(* IEC 61131-3 sources: Lasal/CPU_5344_V01/Class/MillPlanes, 1 file *)

(* ---- MillPlanes.st ---- *)
(*!
<Class
	Name               = "MillPlanes"
	Revision           = "0.0"
	RealtimeTask       = "false"
	CyclicTask         = "false"
	BackgroundTask     = "false"
	Sigmatek           = "false"
	OSInterface        = "false"
	HighPriority       = "false"
	Automatic          = "false"
	UpdateMode         = "Prescan"
	SharedCommandTable = "true"
	Objectsize         = "(450,120)">
	<Channels>
		<Server Name="ClassSvr" Visualized="false" Initialize="false" WriteProtected="true" Retentive="false"/>
		<Server Name="firstIdx" Visualized="true" Initialize="false" WriteProtected="false" Retentive="false"/>
		<Client Name="Line1" Required="true" Internal="true"/>
		<Client Name="Line2" Required="true" Internal="true"/>
		<Client Name="Line3" Required="true" Internal="true"/>
		<Client Name="Line4" Required="true" Internal="true"/>
		<Client Name="Line5" Required="true" Internal="true"/>
		<Client Name="Line6" Required="true" Internal="true"/>
	</Channels>
	<Network Name="MillPlanes">
		<!-- List of Components in this network -->
		<Components>
			<Object
				Name       = "Line1"
				Class      = "MillPlane"
				Position   = "(150,270)"
				Visualized = "true">
				<Channels>
					<Server Name="amount"/>
					<Server Name="ClassSvr"/>
					<Server Name="depth"/>
					<Server Name="feedRate"/>
					<Server Name="firsIdx"/>
					<Server Name="lowerRate"/>
					<Server Name="rnr"/>
				</Channels>
			</Object>
			<Object
				Name       = "Line2"
				Class      = "MillPlane"
				Position   = "(690,270)"
				Visualized = "true">
				<Channels>
					<Server Name="amount"/>
					<Server Name="ClassSvr"/>
					<Server Name="depth"/>
					<Server Name="feedRate"/>
					<Server Name="firsIdx"/>
					<Server Name="lowerRate"/>
					<Server Name="rnr"/>
				</Channels>
			</Object>
			<Object
				Name       = "Line3"
				Class      = "MillPlane"
				Position   = "(1230,270)"
				Visualized = "true">
				<Channels>
					<Server Name="amount"/>
					<Server Name="ClassSvr"/>
					<Server Name="depth"/>
					<Server Name="feedRate"/>
					<Server Name="firsIdx"/>
					<Server Name="lowerRate"/>
					<Server Name="rnr"/>
				</Channels>
			</Object>
			<Object
				Name       = "Line4"
				Class      = "MillPlane"
				Position   = "(1770,270)"
				Visualized = "true">
				<Channels>
					<Server Name="amount"/>
					<Server Name="ClassSvr"/>
					<Server Name="depth"/>
					<Server Name="feedRate"/>
					<Server Name="firsIdx"/>
					<Server Name="lowerRate"/>
					<Server Name="rnr"/>
				</Channels>
			</Object>
			<Object
				Name       = "Line5"
				Class      = "MillPlane"
				Position   = "(2340,270)"
				Visualized = "true">
				<Channels>
					<Server Name="amount"/>
					<Server Name="ClassSvr"/>
					<Server Name="depth"/>
					<Server Name="feedRate"/>
					<Server Name="firsIdx"/>
					<Server Name="lowerRate"/>
					<Server Name="rnr"/>
				</Channels>
			</Object>
			<Object
				Name       = "Line6"
				Class      = "MillPlane"
				Position   = "(2910,270)"
				Visualized = "true">
				<Channels>
					<Server Name="amount"/>
					<Server Name="ClassSvr"/>
					<Server Name="depth"/>
					<Server Name="feedRate"/>
					<Server Name="firsIdx"/>
					<Server Name="lowerRate"/>
					<Server Name="rnr"/>
				</Channels>
			</Object>
		</Components>
		<Comments>
		</Comments>
		<!-- List of Connections in this network -->
		<Connections>
			<Connection Source="this.Line1" Destination="Line1.ClassSvr"/>
			<Connection Source="this.Line2" Destination="Line2.ClassSvr"/>
			<Connection Source="this.Line3" Destination="Line3.ClassSvr"/>
			<Connection Source="this.Line4" Destination="Line4.ClassSvr"/>
			<Connection Source="this.Line5" Destination="Line5.ClassSvr"/>
			<Connection Source="this.Line6" Destination="Line6.ClassSvr"/>
		</Connections>
		<!-- Headerfiles -->
		<Options>
		</Options>
	</Network>
</Class>
*)
MillPlanes : CLASS
  //Servers:
	ClassSvr 	: SvrChCmd_DINT;
	firstIdx 	: SvrCh_DINT;
  //Clients:
	Line2 	: CltChCmd_MillPlane;
	Line3 	: CltChCmd_MillPlane;
	Line6 	: CltChCmd_MillPlane;
	Line5 	: CltChCmd_MillPlane;
	Line1 	: CltChCmd_MillPlane;
	Line4 	: CltChCmd_MillPlane;
  //Variables:
		actPtr 	: ^strMillRecipe;
  //Functions:

	FUNCTION VIRTUAL GLOBAL Init;

	FUNCTION GLOBAL WritePtrs
		VAR_INPUT
			ptr 	: ^strMillRecipe;
		END_VAR;

	FUNCTION VIRTUAL GLOBAL firstIdx::Write
		VAR_INPUT
			input (EAX) 	: DINT;
		END_VAR
		VAR_OUTPUT
			result (EAX) 	: DINT;
		END_VAR;
  //Tables:
	FUNCTION @STD
		VAR_OUTPUT
			ret_code	: CONFSTATES;
		END_VAR;
	FUNCTION GLOBAL TAB @CT_;
END_CLASS;

#pragma using MillPlane

FUNCTION GLOBAL MillPlanes::WritePtrs
	VAR_INPUT
		ptr 	: ^strMillRecipe;
	END_VAR

  actPtr := ptr;

  firstIdx.Write(input:=0);

END_FUNCTION

FUNCTION VIRTUAL GLOBAL MillPlanes::firstIdx::Write
	VAR_INPUT
		input (EAX) 	: DINT;
	END_VAR
	VAR_OUTPUT
		result (EAX) 	: DINT;
	END_VAR

	firstIdx := input;

  if firstIdx >= 0 & firstIdx < (CMAXMILLPLANESINRECIPE) & actPtr<> NIL then
    Line1.WritePtr(iptr:=#actPtr^.planes[firstIdx]);
    Line1.rnr := firstIdx + 1;

//    Line2.WritePtr(iptr:=#actPtr^.planes[firstIdx+1]);
//    Line2.rnr := firstIdx + 2;
//
//    Line3.WritePtr(iptr:=#actPtr^.planes[firstIdx+2]);
//    Line3.rnr := firstIdx +3;
//
//    Line4.WritePtr(iptr:=#actPtr^.planes[firstIdx+3]);
//    Line4.rnr := firstIdx +4;
//
//    Line5.WritePtr(iptr:=#actPtr^.planes[firstIdx+4]);
//    Line5.rnr := firstIdx +5;
//
//    Line6.WritePtr(iptr:=#actPtr^.planes[firstIdx+5]);
//    Line6.rnr := firstIdx +6;

  else
    result := ACCESS_DENIED;
    if firstIdx> 0 then
      firstIdx-=1;
    else
      firstIdx+=1;
    end_if;
  end_if;
    result := firstIdx;

END_FUNCTION

FUNCTION VIRTUAL GLOBAL MillPlanes::Init
  // op startup firstidx writen om alles een rnr te geven
  firstIdx.Write(input:=0);

END_FUNCTION
